TYPE UDT_OeeHmi_RD :
STRUCT
start                  : BOOL; // 开始
end                    : BOOL; // 结束
clear                  : BOOL; // 清零
scheduledDown          : BOOL; // 计划停止
startTimeDisplay       : BOOL; // 开始时刻显示
endTimeDisplay         : BOOL; // 结束时刻显示
goodValue              : DINT; // 良品数量
badValue               : DINT; // 不良品数量
totalValue             : DINT; // 总数量
availability           : REAL; // 可用率
performance            : REAL; // 性能指数
quality                : REAL; // 质量指数
oee                    : REAL; // 综合效率
startTime              : ARRAY[0..6] OF INT; // 开始时刻
endTime                : ARRAY[0..6] OF INT; // 结束时刻
totalTime              : UDT_DayTime_RD; // 总时间
productiveTime         : UDT_DayTime_RD; // 生产时间
downTime               : UDT_DayTime_RD; // 计划停机时间
runtime                : UDT_DayTime_RD; // 运行时间
standbyTime            : UDT_DayTime_RD; // 待机时间
failureTime            : UDT_DayTime_RD; // 故障时间
failureCount           : UINT; // 故障次数
number                 : INT; // 编号

END_STRUCT
END_TYPE

(* stored: Version 1.1.0.1, ProductVersion 3.1.4024.12
   DUT UDT_OeeHmi_RD: Id {e624ca82-3e80-4572-8d42-bc2a2801fc41} *)
